{attribute 'linkalways'} 
{attribute 'no_explicit_call' := 'This FB is a CLASS and must be accessed using methods or properties'}
{attribute 'enable_dynamic_creation'}
FUNCTION_BLOCK FINAL MAX_ULINT EXTENDS Node
VAR
	in1 : _ULINT(0);
	in2 : _ULINT(0);
	out : _ULINT(0);
END_VAR

METHOD PUBLIC Clone : I_Node
VAR
	pNode : POINTER TO MAX_ULINT;
END_VAR
pNode := __NEW(MAX_ULINT);
Clone := pNode^;
END_METHOD

METHOD FB_init : BOOL
VAR_INPUT
	bInitRetains : BOOL; // if TRUE, the retain variables are initialized (warm start / cold start)
	bInCopyCode : BOOL;  // if TRUE, the instance afterwards gets moved into the copy code (online change)
END_VAR
AddInput('in1',THIS^.in1);
AddInput('in2',THIS^.in2);
AddOutput('out', THIS^.out);
END_METHOD

METHOD PROTECTED OnExecute
VAR
END_VAR
out.Value := MAX(in1.Value, in2.Value);
END_METHOD

END_FUNCTION_BLOCK

(* stored: Version 1.1.0.1, ProductVersion 3.1.4024.15
   POU MAX_ULINT: Id {0e0a0aec-5ad2-458d-a9eb-8d6622910ad6}, SpecialFunc None
   Folder Constructor: Id {a2cc9e05-e4fb-47bd-9684-f50fbb21c6af}
   Method Clone: Id {07d65c00-971b-4eff-8ea8-1d7f2d21d727}
   Method FB_init: Id {c0b8a27b-6654-4c7d-8df8-3f1f004208ea}
   Method OnExecute: Id {a18135cf-7e54-4457-95c3-899efc707220} *)
